FUNCTION_BLOCK ConveyorCTLMulticast (* Basic Function Block Type forMulticast *)
  (* Standard: 61499-2 *)
  (* Version 0.2, 2003-12-04, JHC, Rockwell Automation, Renamed for better indexing. *)
  (* Version 0.1, 2002-11-05, JHC, Rockwell Automation, Corrected missing ST element in Algorithm REQ. *)
  (* Version 0.0, 2000-05-30, JHC, Rockwell Automation *)
  (* Compiler header: package fb.rt.cs725; *)
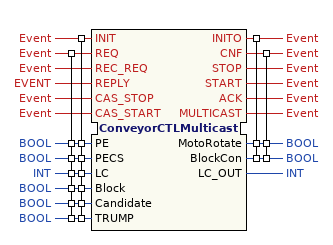
  EVENT_INPUT
    INIT WITH PE, Block, Candidate, PECS, LC, TRUMP; (* Initialization Request *)
    REQ WITH PE, Block, Candidate, PECS, LC, TRUMP; (* Normal Execution Request *)
    REC_REQ;
    REPLY : EVENT;
    CAS_STOP;
    CAS_START;
  END_EVENT
  EVENT_OUTPUT
    INITO WITH MotoRotate, BlockCon; (* Initialization Confirm *)
    CNF WITH MotoRotate, BlockCon; (* Execution Confirmation *)
    STOP;
    START;
    ACK;
    MULTICAST;
  END_EVENT
  VAR_INPUT
    PE : BOOL; (* Input event qualifier *)
    PECS : BOOL;
    LC : INT;
    Block : BOOL;
    Candidate : BOOL;
    TRUMP : BOOL;
  END_VAR
  VAR_OUTPUT
    MotoRotate : BOOL; (* Output event qualifier *)
    BlockCon : BOOL;
    LC_OUT : INT;
  END_VAR
  VAR
    lastPE : BOOL := 1;
    lastBlock : BOOL := 0;
    LAM_CLOCK : INT;
    HAS_TOKEN : BOOL;
  END_VAR
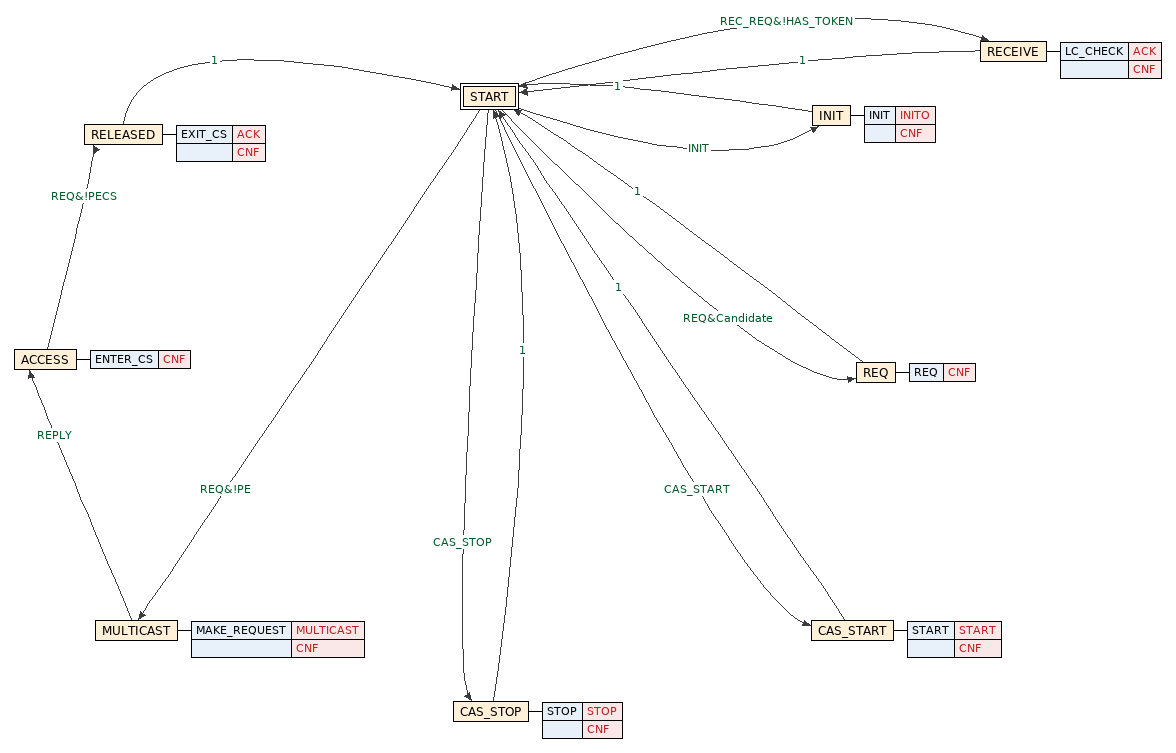
  EC_STATES
    START; (* Initial State *)
    INIT : INIT -> INITO, -> CNF; (* Initialization *)
    REQ : REQ -> CNF; (* Normal execution *)
    CAS_START : START -> START, -> CNF;
    CAS_STOP : STOP -> STOP, -> CNF;
    MULTICAST : MAKE_REQUEST -> MULTICAST, -> CNF; (* When bag is detected, send requests *)
    ACCESS : ENTER_CS -> CNF;
    RELEASED : EXIT_CS -> ACK, -> CNF;
    RECEIVE : LC_CHECK -> ACK, -> CNF;
  END_STATES
  EC_TRANSITIONS
    START TO INIT := INIT;
    INIT TO START := 1;
    START TO REQ := REQ&Candidate;
    REQ TO START := 1;
    START TO CAS_START := CAS_START;
    CAS_START TO START := 1;
    START TO CAS_STOP := CAS_STOP;
    CAS_STOP TO START := 1;
    START TO MULTICAST := REQ&!PE;
    MULTICAST TO ACCESS := REPLY;
    ACCESS TO RELEASED := REQ&!PECS;
    RELEASED TO START := 1;
    START TO RECEIVE := REC_REQ&!HAS_TOKEN;
    RECEIVE TO START := 1;
  END_TRANSITIONS
  ALGORITHM INIT IN ST: (* Initialization algorithm *)
MotoRotate := TRUE;
Block := FALSE;

System.out.println(this + " " + MotoRotate);
System.out.println(MotoRotate);
  END_ALGORITHM
  ALGORITHM REQ IN ST: (* Normally executed algorithm *)
System.out.println(this +  " -> Candidate" + Candidate);
IF Candidate THEN
IF lastPE !:= PE THEN
IF NOT PE THEN
BlockCon:= TRUE;
System.out.println("BlockCon = true");
ELSE
BlockCon:=FALSE;
System.out.println("BlockCon = false");
END_IF
lastPE := PE;
END_IF
IF lastBlock !:= Block THEN
IF Block THEN
STOP.serviceEvent(this);
MotoRotate := FALSE;
System.out.println("Cas Stop");
ELSE
START.serviceEvent(this);
MotoRotate := TRUE;
System.out.println("Cas Start");
END_IF
lastBlock := Block;
END_IF
END_IF
  END_ALGORITHM
  ALGORITHM START IN ST:
MotoRotate:=TRUE;
System.out.println(this + " Start " + MotoRotate);

System.out.println("Start " + MotoRotate);
  END_ALGORITHM
  ALGORITHM STOP IN ST:
MotoRotate := FALSE;
System.out.println(this + " Stop " + MotoRotate);

System.out.println("Stop " + MotoRotate);
  END_ALGORITHM
  ALGORITHM MAKE_REQUEST IN Java:
LAM_CLOCK.value++;
LC_OUT.value = LAM_CLOCK.value;
MotoRotate.value = false;
System.out.printf("[MULTICAST] Request, LC:%d%n", LAM_CLOCK);
  END_ALGORITHM
  ALGORITHM ENTER_CS IN Java:
HAS_TOKEN.value = true;
MotoRotate.value = true;
System.out.println("[MULTICAST] Enter CS");
  END_ALGORITHM
  ALGORITHM EXIT_CS IN Java:
HAS_TOKEN.value = true;
System.out.println("[MULTICAST] Exit CS");
  END_ALGORITHM
  ALGORITHM LC_CHECK IN Java:
System.out.println("[MULTICAST] Received request");
if (LC.value > LAM_CLOCK.value) {
LAM_CLOCK.value = LC.value;
System.out.println("[MULTICAST] LC Updated");
}
  END_ALGORITHM
END_FUNCTION_BLOCK
